FUNCTION_BLOCK FB_12PVICI_EPS
VAR_INPUT
    iAdress : INT;
END_VAR
VAR_OUTPUT
    bAllPortsLocked : BOOL;
    bExternalLock : BOOL;
END_VAR
VAR_IN_OUT
    aPortEPS : ARRAY [*] OF DUT_VICI_PORT_EPS; // EPS for each port.
END_VAR
VAR
    fbNporValve : FB_ViciValve;
    iNumPorts : INT := 12;

    {attribute 'pytmc' := '
        pv: iReqPos
        io: io
     '}
    iReqPos : INT;
    {attribute 'pytmc' := '
        pv: SampleNames
        io: io
     '}
    stSampleNames : ST_12ViciValveSampleNames;

    // EPS
    {attribute 'pytmc' := '
    pv: iEPSPORT
    io: o
    '}
    iNewPort : INT;
    {attribute 'pytmc' := '
    pv: fbEPS
    io: o
    '}
    fbViciEPS : FB_VICI_EPS;

    {attribute 'pytmc' := 'pv: bOVRD_MODE'}
    bEPS_Override : BOOL := FALSE;

    {attribute 'pytmc' := 'pv: bOVRD_COUNTDOWN'}
    tEPS_TimerCountDown : STRING := TIME_TO_STRING(T#0s);
END_VAR

iReqPos := LIMIT(1,iReqPos, iNumPorts); // KEEP EPS array index within bounds

fbViciEPS(aPortEPS := aPortEPS,
    iReqPort := iReqPos,
    iPrevPort := iNewPort,
    bOverride := bEPS_Override,
    iNumPorts := iNumPorts,
    bExternalLockSignal => bExternalLock,
    bAllPortsLocked => bAllPortsLocked,
    iNewPortPos => iNewPort,
    tEPS_TimerCountDown => tEPS_TimerCountDown);

iReqPos := iNewPort; // Updat iReqPos PV  to be the safe port, otherwise when EPS is cleared the requested port would automatically change.

fbNporValve(iAddress := iAdress,
    iNumOfPorts := iNumPorts,
    iReqPos := iNewPort);

END_FUNCTION_BLOCK

(* stored: Version 1.1.0.1, ProductVersion 3.1.4024.12
   POU FB_12PVICI_EPS: Id {31d89ef3-b073-4080-b347-efa36ca070a2}, SpecialFunc None *)
